INTERFACE I_Observable  EXTENDS __SYSTEM.IQueryInterface

METHOD add_observer : BOOL
VAR_INPUT
	observer : I_Observer;
END_VAR
END_METHOD

PROPERTY error_id : HRESULT
GET
END_GET
SET
END_SET
END_PROPERTY

METHOD notify_observers : BOOL
END_METHOD

METHOD remove_observer : BOOL
VAR_INPUT
	observer : I_Observer;
END_VAR
END_METHOD

END_INTERFACE

(* stored: Version 1.1.0.1, ProductVersion 3.1.4026.13
   Itf I_Observable: Id {92b993e2-e7c7-4e67-97d7-3ed763275f90}
   Method add_observer: Id {bd642e2f-5d27-4e66-9f33-1a521b718282}
   Property error_id: Id {739f0bef-5b2f-442e-b61b-84f0fa9315ae}
   Get Get: Id {6f7cbb61-27f2-4b23-91f9-81214f215639}
   Set Set: Id {2773258f-ffde-4726-b18c-291029fae65b}
   Method notify_observers: Id {54582a89-72cc-477c-a748-1b58ee3b7a78}
   Method remove_observer: Id {4e028d00-22a0-48ff-b97c-9c0590df9e11} *)
